// Mitsubishi GX Works2 project: Time n Count   PLC: FX3U/FX3UC

PROGRAM MAIN
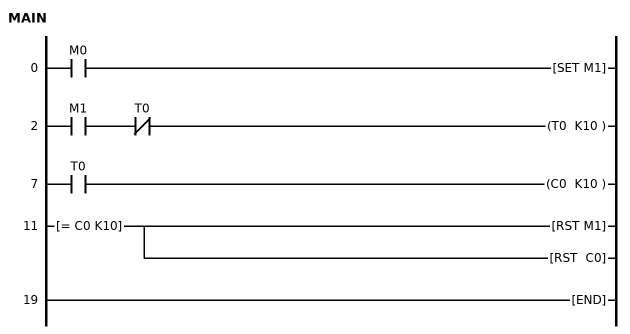
0     LD      M0
      SET     M1
2     LD      M1
      ANI     T0
      OUT     T0 K10
7     LD      T0
      OUT     C0 K10
11    LD=     C0 K10
      RST     M1
      RST     C0
19    END
END_PROGRAM
